Universal Robots PolyScope program: 20240817_balloon.urp

Program 20240817_balloon (installation=default directory=/programs/servoj createdIn=5.13.1 lastSavedIn=5.13.1 robotSerialNumber=20195380017)
Calibrated DH parameters: a=[-0.000005, -0.241897, -0.163857, -0.000004, -0.000042, 0]; d=[0.15198, 4.092034, -18.51686, 14.555458, 0.085328, 0.092191]; alpha=[1.570113, -0.007378, -0.009451, 1.571508, -1.571142, 0]; deltaTheta=[-0.000001, -0.124164, 0.818102, -0.693964, 0.000084, 0]
InitVariablesNode
Robot Program (runOnlyOnce=true)
  Popup Message (haltProgram=false message=please ensure the state inputType=Text)
  Wait Sleep waitTime=0.8
  SuppressedNode
    Halt
  Loop Counting (count=10) loopVariable(name=循环_2)
    MoveL speed 100 mm/s, acceleration 600 mm/s^2 (useActiveTCP=true) feature=Base
      Waypoint 路点_1: motionParameters(jointSpeed=1.047198 jointAcceleration=1.396263 cartesianSpeed=0.12 cartesianAcceleration=0.8); TCP in base x=-4.702 y=-269.784 z=97.715 mm, rx=-2.1972 ry=2.2419 rz=0.006 rad; joints [-58.248, -76.106, -95.761, -98.357, 89.817, -56.231] deg; TCP offset x=1.06 y=22.52 z=227.92 mm, rx=0 ry=0 rz=0 rad
      Waypoint 路点_3: motionParameters(jointSpeed=1.047198 jointAcceleration=1.396263 cartesianSpeed=0.06 cartesianAcceleration=0.6); TCP in base x=-4.699 y=-425.554 z=97.725 mm, rx=-2.1972 ry=2.2419 rz=0.006 rad; joints [-70.171, -117.706, -48.295, -104.241, 89.516, -68.19] deg
        Until EXPRESSION (allowActions=true deceleration=2) ExpressionBranch=tmp[0]≥1
          Wait Sleep waitTime=0.5
Thread Thread_1 (runOnlyOnce=false)
  tmp := p[0,0,0,0,0,0]
  Loop Forever
    Script file /programs/pose_register.script
      | tmp[0]=read_input_float_register(0)
      | tmp[1]=read_input_float_register(1)
      | tmp[2]=read_input_float_register(2)
      | tmp[3]=read_input_float_register(3)
      | tmp[4]=read_input_float_register(4)
      | tmp[5]=read_input_float_register(5)
    Script: sync()
